FUNCTION_BLOCK Integrator
VAR_INPUT
	x : REAL;
	h : REAL;
END_VAR
VAR_OUTPUT
	y : REAL;
END_VAR
VAR
	xm : REAL;
	ym : REAL;
END_VAR

y := xm * h + ym;
ym := y;
xm : = x;

END_FUNCTION_BLOCK

(* stored: Version 1.1.0.1, ProductVersion 3.1.4024.13
   POU Integrator: Id {11aae5db-9c23-4224-ac47-adc1a4f2d2d4}, SpecialFunc None *)
